(* PLC project Unnamed, Unknown Unnamed 1 *)
(* stored: creationDateTime 2025-06-13T16:30:15, modificationDateTime 2025-06-13T18:40:06 *)

PROGRAM part3
  VAR
    state : UINT := 0;
    wait_for_request : UINT := 0;
    wait_for_traffic : UINT := 1;
    slow_cars : UINT := 2;
    ped_xing : UINT := 3;
    all_red : UINT := 4;
  END_VAR
  VAR
    car_sensor AT %IX0.0 : BOOL;
    ped_button AT %IX0.1 : BOOL;
    car_red AT %QX0.0 : BOOL;
    car_yellow AT %QX0.1 : BOOL;
    car_green AT %QX0.2 : BOOL;
    ped_red AT %QX0.3 : BOOL;
    ped_green AT %QX0.4 : BOOL;
  END_VAR
  VAR
    TON0 : TON;
    yellow_delay : TIME := T#3s;
    ped_xing_delay : TIME := T#15s;
    all_red_delay : TIME := T#1s;
    TON1 : TON;
    TON2 : TON;
    waiting_for_request : BOOL := 0;
    waiting_for_traffic : BOOL := 0;
    slowing_cars : BOOL := 0;
    peds_xing : BOOL := 0;
    turning_all_red : BOOL := 0;
  END_VAR

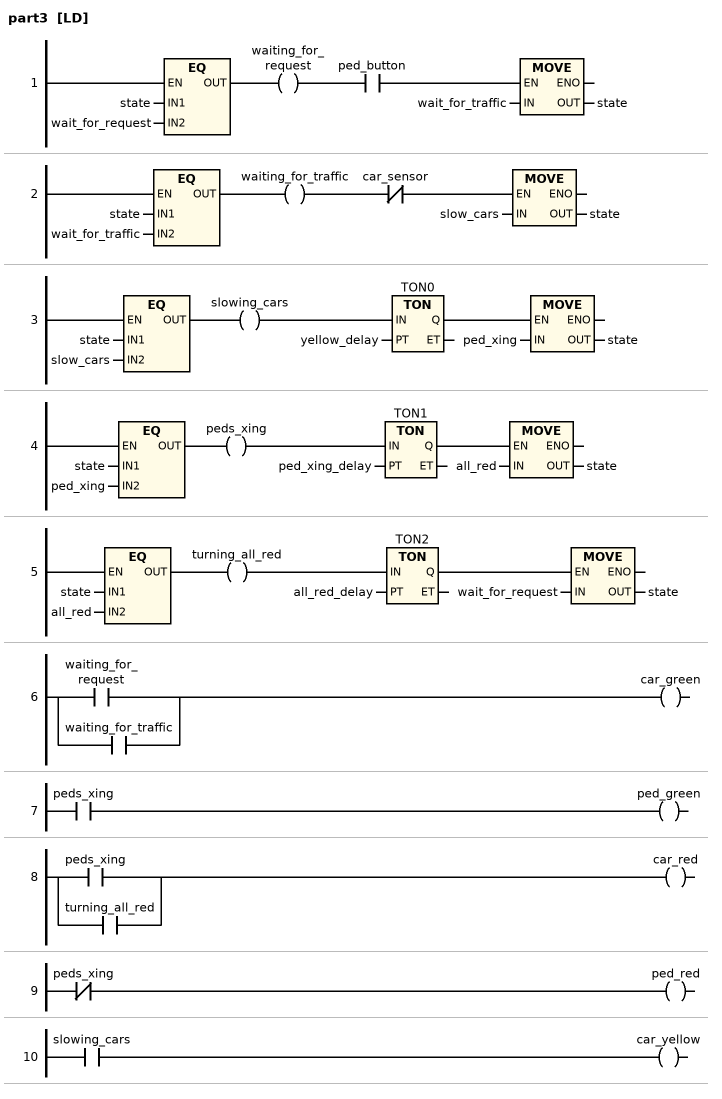
(* LD diagram, written out as Structured Text *)
IF state = wait_for_request AND ped_button THEN state := wait_for_traffic; END_IF;
IF state = wait_for_traffic AND NOT car_sensor THEN state := slow_cars; END_IF;
TON0(IN := state = slow_cars, PT := yellow_delay);
IF TON0.Q THEN state := ped_xing; END_IF;
TON1(IN := state = ped_xing, PT := ped_xing_delay);
IF TON1.Q THEN state := all_red; END_IF;
TON2(IN := state = all_red, PT := all_red_delay);
IF TON2.Q THEN state := wait_for_request; END_IF;
waiting_for_request := state = wait_for_request;
waiting_for_traffic := state = wait_for_traffic;
slowing_cars := state = slow_cars;
peds_xing := state = ped_xing;
turning_all_red := state = all_red;
car_green := waiting_for_request OR waiting_for_traffic;
ped_green := peds_xing;
car_red := peds_xing OR turning_all_red;
ped_red := NOT peds_xing;
car_yellow := slowing_cars;
END_PROGRAM

CONFIGURATION Config0
  RESOURCE Res0 ON PLC
    TASK task0(INTERVAL := T#20ms, PRIORITY := 0);
    PROGRAM instance0 WITH task0 : part3;
  END_RESOURCE
END_CONFIGURATION
